PROGRAM MAIN
VAR
	X_Axis			: AXIS_REF;
	Y_Axis			: AXIS_REF;
	Z_Axis			: AXIS_REF;
END_VAR

END_PROGRAM

(* stored: Version 1.1.0.1, ProductVersion 3.1.4024.10
   POU MAIN: Id {0ed01888-47ce-42c9-9b1b-67fc9476a6f3}, SpecialFunc None *)
